FUNCTION_BLOCK FB_AutoClock
VAR_INPUT
	fStart : BOOL;
	fRunning : BOOL;
	fCycle : LREAL;
END_VAR
VAR_OUTPUT
	fTime : LREAL;
END_VAR
VAR
END_VAR


IF NOT(fStart) OR NOT(fRunning) THEN
	fTime := 0.0;
ELSIF fStart AND fRunning THEN
	fTime := fTime + fCycle;		
END_IF

END_FUNCTION_BLOCK

(* stored: Version 1.1.0.1, ProductVersion 3.1.4024.12
   POU FB_AutoClock: Id {7377a5f2-2bb2-4a99-a851-408be3481e91}, SpecialFunc None *)
